PROGRAM Q6
VAR
	// Parts present?
	partA : BOOL := FALSE;
	partB : BOOL := FALSE;	
	
	// Button pressed?
	button : BOOL := FALSE;
	
	// Running operation
	TON_0: TON;
	time_ext : TIME := T#1S;
	extend : BOOL := FALSE;
	
	// Transition flags
	start: BOOL := FALSE;
	complete : BOOL := FALSE;
	
END_VAR

// BSOD recovery @ 1447hrs
// BSOD recovery @ 1519hrs - currently running at 1.2 crashes per hour!

// Not fully working yet - those crashes cost about five minutes each!

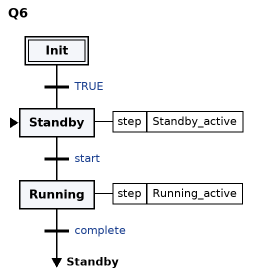
INITIAL_STEP Init:
END_STEP
TRANSITION FROM Init TO Standby
    := TRUE;
END_TRANSITION
STEP Standby:
    Standby_active(N);  // step action
END_STEP
TRANSITION FROM Standby TO Running
    := start;
END_TRANSITION
STEP Running:
    Running_active(N);  // step action
END_STEP
TRANSITION FROM Running TO Standby
    := complete;
END_TRANSITION

ACTION Running_active:
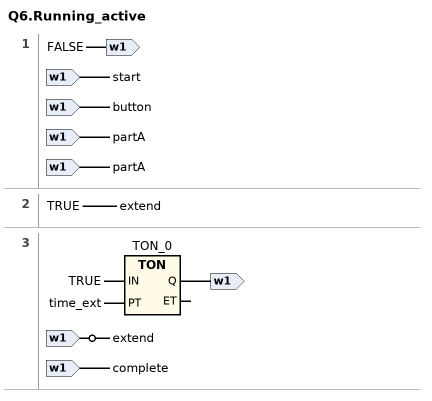
// NETWORK 1
start := FALSE;
button := FALSE;
partA := FALSE;
partA := FALSE;

// NETWORK 2
extend := TRUE;

// NETWORK 3
TON_0(IN := TRUE, PT := time_ext); // TON
extend := NOT TON_0.Q;
complete := TON_0.Q;
END_ACTION

ACTION Standby_active:
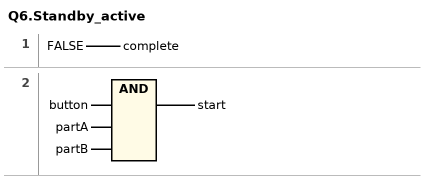
// NETWORK 1
complete := FALSE;

// NETWORK 2
start := button AND partA AND partB;
END_ACTION

END_PROGRAM

(* stored: Version 1.1.0.1, ProductVersion 3.1.4024.12
   POU Q6: Id {db4561dc-87ee-4342-acad-72836d5ab132}, SpecialFunc None
   Action Running_active: Id {87f1ad34-04b3-4655-96fd-5811ce3b0389}
   Action Standby_active: Id {88ff75fb-ce67-4216-b530-7c776a27c9dd} *)
